// TIA Portal V17 export
// export: Created 2024-09-02T12:49:54.1965258Z, ExportSetting WithDefaults, DisplayName Totally Integrated Automation Portal, DisplayVersion V17, DisplayName TIA Portal Openness, DisplayVersion V17, DisplayName TIA Portal Version Control Interface, DisplayVersion V17, DisplayName STEP 7 Professional, DisplayVersion V17, DisplayName STEP 7 Safety, DisplayVersion V17, DisplayName WinCC Professional, DisplayVersion V17
DATA_BLOCK "AnwDB_Data_to_Safety"   // DB7005
{ S7_Optimized_Access := 'TRUE'; DB_Accessible_From_OPC_UA := 'FALSE' }
AUTHOR : VAF
VERSION : 0.1
// stored: AutoNumber false, DBAccessibleFromOPCUA false, IsOnlyStoredInLoadMemory false, IsRetainMemResEnabled false, IsWriteProtectedInAS false, MemoryReserve 0
   VAR
      "Media On_2" : Bool;
      "Media On_1" : Bool;
      "Fault acknowledge_2" : Bool;
      "Fault acknowledge_1" : Bool;
      ProtectiveCircuitAcknowledge_2 : Bool;
      ProtectiveCircuitAcknowledge_1 : Bool;
      AssembliesAcknowledge_2 : Bool;
      AssembliesAcknowledge_1 : Bool;
      "res0.4" : Bool;
      "res0.5" : Bool;
      "res0.6" : Bool;
      "res0.7" : Bool;
      LampTest : Bool;
      "res1.1" : Bool;
      "res1.2" : Bool;
      "res1.3" : Bool;
      "res1.4" : Bool;
      "res1.5" : Bool;
      "res1.6" : Bool;
      "res1.7" : Bool;
      SafetyDoorUnlock : Array[0..16] of Bool;
   END_VAR
BEGIN
END_DATA_BLOCK
